(* PLC project poST.project, poSTIDE *)
(* stored: creationDateTime 2021-08-31T00:00:00.000000 *)

FUNCTION MOVE : ANY
  VAR_INPUT
    in : ANY;
  END_VAR

END_FUNCTION
